% RSLogix 500 project LAB 2 Q4 ROBO_done.RSS, saved by version 8.40.00.08 %
PROJECT "UNTITLED"    % processor: type code 162 %

PROGRAM FILES
  LAD 2   11 rungs

DATA FILES
  S2 STATUS  83 elements
  B3 BINARY  1 elements
  T4 TIMER  1 elements
  C5 COUNTER  1 elements
  R6 CONTROL  1 elements
  N7 INTEGER  1 elements
  F8 FLOAT  1 elements

LADDER 2
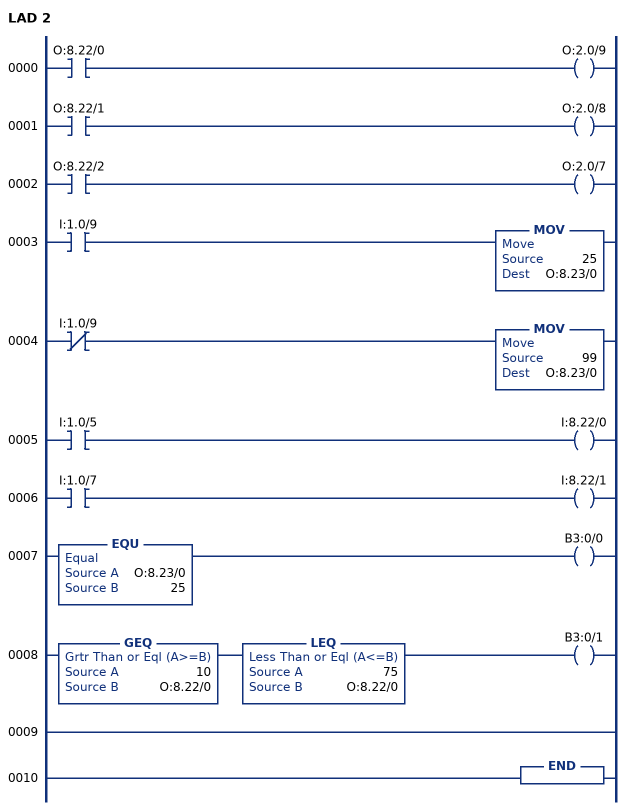
% Rung: 0 %  % edit flag set %
SOR XIC O:8.22/0 OTE O:2.0/9 EOR
% Rung: 1 %  % edit flag set %
SOR XIC O:8.22/1 OTE O:2.0/8 EOR
% Rung: 2 %  % edit flag set %
SOR XIC O:8.22/2 OTE O:2.0/7 EOR
% Rung: 3 %  % edit flag set %
SOR XIC I:1.0/9 MOV 25 O:8.23/0 EOR
% Rung: 4 %  % edit flag set %
SOR XIO I:1.0/9 MOV 99 O:8.23/0 EOR
% Rung: 5 %  % edit flag set %
SOR XIC I:1.0/5 OTE I:8.22/0 EOR
% Rung: 6 %  % edit flag set %
SOR XIC I:1.0/7 OTE I:8.22/1 EOR
% Rung: 7 %  % edit flag set %
SOR EQU O:8.23/0 25 OTE B3:0/0 EOR
% Rung: 8 %  % edit flag set %
SOR GEQ 10 O:8.22/0 LEQ 75 O:8.22/0 OTE B3:0/1 EOR
% Rung: 9 %  % edit flag set %
SOR EOR
% Rung: 10 %
SOR END EOR
